TYPE T_Ctrl_Info :
STRUCT
	///name of controller instance
	strName: STRING(80);
	///class of controller
	strType: STRING(80);
	///unique controller instance identification number
	intCtrlId: INT;
	///unique identification number of parent controller instance
	intParentCtrlId: INT;
	///all inputs valid -> init done
	bolInitDone: BOOL;
	///Childs
	p_afbChild: ARRAY[0..Base_Const.cMaxNrOfChilds] OF POINTER TO BYTE;
	///common interface array of childs
	p_aCIf: ARRAY[0..Base_Const.cMaxNrOfChilds] OF POINTER TO T_Ctrl_CIf;
END_STRUCT
END_TYPE

(* stored: Version 1.1.0.1, ProductVersion 3.1.0.18
   DUT T_Ctrl_Info: Id {8e469935-d33b-4e57-b8fe-b5aa8dfa713d} *)
